{attribute 'enable_dynamic_creation'}	
{attribute 'no_explicit_call' := 'do not call this function block directly'} 
FUNCTION_BLOCK ABSTRACT Exception EXTENDS Object IMPLEMENTS IException
VAR
	_Fatal : BOOL; 	
	_SourceNamespaceName : STRING;
	_SourceClassName : STRING;
	_SourceMethodName : STRING;
	_SourcePosition : STRING;
	_LocalTimestamp : DATE_AND_TIME;	
	_UtcTimestamp : DATE_AND_TIME;	
END_VAR
VAR CONSTANT
	PATH_DELIMITER : WSTRING(1) := ".";
	UNSPECIFIED_METHOD : WSTRING(20) := "<unspecified method>";
	TIME_PREFIX : WSTRING(4) := " at ";
	SOURCE_PREFIX : WSTRING(4) := " in ";
	ERROR_CODE_PREFIX : WSTRING(13) := ", error code ";	
	LINE_NUMBER_PREFIX : WSTRING(13) := " line ";	
	INNER_MESSAGE_PREFIX : WSTRING(4) := " -> ";
END_VAR

METHOD PROTECTED AppendProgramOrganizationUnitFullName
VAR_IN_OUT CONSTANT
	stringBuilder : WideStringBuilder;
END_VAR
stringBuilder
	.AppendIf(_SourceNamespaceName, SourceNamespaceName <> '')
	.AppendStringIf(PATH_DELIMITER, SourceNamespaceName <> '')
	.AppendIf(_SourceClassName, SourceClassName <> '')
	.AppendStringIf(PATH_DELIMITER, SourceClassName <> '')
	.AppendIf(_SourceMethodName, SourceMethodName <> '')
	.AppendStringIf(UNSPECIFIED_METHOD, SourceMethodName = '');
END_METHOD

METHOD PROTECTED AppendSourceDescription
VAR_IN_OUT CONSTANT
	stringBuilder : WideStringBuilder;
END_VAR
AppendProgramOrganizationUnitFullName(stringBuilder);

stringBuilder
	.AppendStringIf(LINE_NUMBER_PREFIX, SourcePosition <> '')
	.AppendIf(_SourcePosition, SourcePosition <> '');
END_METHOD

METHOD PROTECTED AppendTimestampDescription
VAR_IN_OUT CONSTANT
	stringBuilder : WideStringBuilder;
END_VAR
stringBuilder
	.Append(_LocalTimestamp)
	.AppendString(" (")
	.Append(_UtcTimestamp)
	.AppendString("UTC)");
END_METHOD

METHOD ABSTRACT Clone : IObject
END_METHOD

{attribute 'monitoring' := 'call'}
PROPERTY ABSTRACT Empty : BOOL
GET
END_GET
END_PROPERTY

// Work is not possible after such error
{attribute 'monitoring' := 'call'}
PROPERTY Fatal : BOOL
GET
Fatal := _Fatal;
END_GET
SET // PROTECTED
_Fatal := Fatal;
END_SET
END_PROPERTY

METHOD ABSTRACT GetMessage : ERROR_MESSAGE
VAR_INPUT
	showTimestamp : BOOL := FALSE;
	showSource : BOOL := FALSE;
END_VAR
END_METHOD

METHOD GetSourceDescription : WSTRING(300)
VAR
	stringBuilder : WideStringBuilder;
END_VAR
AppendSourceDescription(stringBuilder);

stringBuilder.AssignToString(GetSourceDescription);
END_METHOD

{attribute 'monitoring' := 'call'}
PROPERTY LocalTimestamp : DATE_AND_TIME
GET
LocalTimestamp := _LocalTimestamp;
END_GET
SET // PROTECTED
_LocalTimestamp := LocalTimestamp;
END_SET
END_PROPERTY

{attribute 'monitoring' := 'call'}
PROPERTY SourceClassName : STRING
GET
SourceClassName := _SourceClassName;
END_GET
SET // PROTECTED
_SourceClassName := SourceClassName;
END_SET
END_PROPERTY

{attribute 'monitoring' := 'call'}
PROPERTY SourceMethodName : STRING
GET
SourceMethodName := _SourceMethodName;
END_GET
SET // PROTECTED
_SourceMethodName := SourceMethodName;
END_SET
END_PROPERTY

{attribute 'monitoring' := 'call'}
PROPERTY SourceNamespaceName : STRING
GET
SourceNamespaceName := _SourceNamespaceName;
END_GET
SET // PROTECTED
_SourceNamespaceName := SourceNamespaceName;
END_SET
END_PROPERTY

{attribute 'monitoring' := 'call'}
PROPERTY SourcePosition : STRING
GET
SourcePosition := _SourcePosition;
END_GET
SET // PROTECTED
_SourcePosition := SourcePosition;
END_SET
END_PROPERTY

{attribute 'monitoring' := 'call'}
PROPERTY UtcTimestamp : DATE_AND_TIME
GET
UtcTimestamp := _UtcTimestamp;
END_GET
SET // PROTECTED
_UtcTimestamp := UtcTimestamp;
END_SET
END_PROPERTY

END_FUNCTION_BLOCK

(* stored: Version 1.1.0.1
   POU Exception: Id {2c867dd1-35d5-4b22-aba9-7dd48de148f5}, SpecialFunc None
   Folder Service members: Id {7fcae734-384a-4348-b662-c86a9b6ee9b5}
   Method AppendProgramOrganizationUnitFullName: Id {8b619731-2c00-46d9-91ce-b530c604c931}
   Method AppendSourceDescription: Id {232ae1fb-919d-444e-a1b1-41423c0a2e61}
   Method AppendTimestampDescription: Id {2603d8b7-93f6-4d37-b896-c4502bdc4dce}
   Method Clone: Id {5ebd59ef-8f06-4536-82ff-256e85b923d6}
   Property Empty: Id {5808a72a-29e6-41ff-a698-14358227f440}
   Get Get: Id {baf9f777-1bbb-46e3-a0e2-7b890beb87c1}
   Property Fatal: Id {c5832d03-a61c-4285-ad48-f70a09db5cc4}
   Get Get: Id {bd66e01d-04bc-4ecf-9bbf-76e999d0693f}
   Set Set: Id {78a9683e-7789-4360-aa2a-0c4ebea628b6}
   Method GetMessage: Id {b01f2e4b-f57f-4a9e-9bb1-0d11fe56eeb6}
   Method GetSourceDescription: Id {4b3d6002-41a8-4524-9636-7a2f25a8d478}
   Property LocalTimestamp: Id {440a2ace-f694-4eeb-8122-2b10d9458da0}
   Get Get: Id {c53a1132-41e2-418b-b336-bd0a0d1f095b}
   Set Set: Id {29a6d1f5-af60-43ea-8bf5-4492964b6fc2}
   Property SourceClassName: Id {b6bf95b3-05bb-41c1-baf2-adec7e4807a2}
   Get Get: Id {da8e8243-9de1-4f25-9aef-7229c118af25}
   Set Set: Id {f9b92e01-f998-4ca4-b6d7-455ed4a82e72}
   Property SourceMethodName: Id {b0b11d8f-b57d-436d-a30b-45c5828bcad7}
   Get Get: Id {430fe027-4455-4395-b14b-1ccf8dd03c14}
   Set Set: Id {9d5e5bf5-fffc-43c7-b803-fd8e6fd15bef}
   Property SourceNamespaceName: Id {69392083-68c6-4dcd-bb09-4e25ac9807d1}
   Get Get: Id {b37bec38-ccba-44a5-adba-4d95aa902bc2}
   Set Set: Id {89292779-957c-4b86-a678-d58842d0ba8f}
   Property SourcePosition: Id {3841f015-137e-4d98-b3a5-a880f1f999fe}
   Get Get: Id {2126c131-19e6-4818-8020-5003129f9123}
   Set Set: Id {5d557cbc-73a7-412c-88fc-e096352966b1}
   Property UtcTimestamp: Id {e428f86e-5f4a-4af4-a349-fca47e15fa8e}
   Get Get: Id {2bb3d289-0f15-49af-b239-4833a8a2dc7b}
   Set Set: Id {8bca7369-3782-4526-91b9-39c4010a000e} *)
